FUNCTION_BLOCK "Main"
VERSION : 0.1
   VAR_INPUT
      in1 : Bool;
      in2 : Bool;
      in3 : Bool;
   END_VAR

   VAR_OUTPUT
      out1 : Bool;
   END_VAR


BEGIN
NETWORK
TITLE =
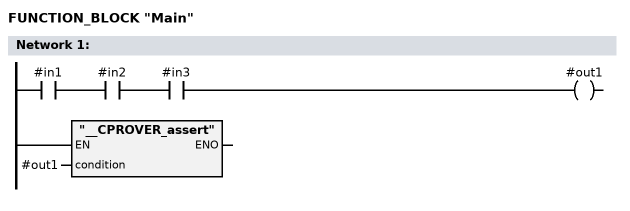
      A #in1;
      A #in2;
      A #in3;
      = #out1;
      CALL "__CPROVER_assert"
      (  condition := #out1
      );

END_FUNCTION_BLOCK

